// TIA Portal V20 export
TYPE "typeSequenceControlNodeHomeCheck"
// stored: Namespace Unit1.Em0
   STRUCT
      partNoGet { ExternalWritable := 'False'} : Bool;
      partGet { ExternalWritable := 'False'} : Bool;
   END_STRUCT;
END_TYPE
